ABB RobotStudio station: comportamiento1.rspag

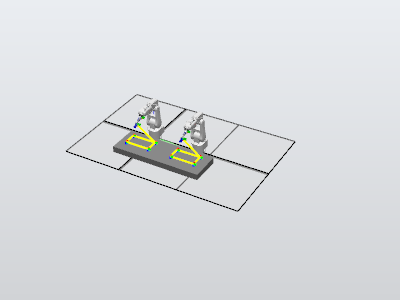
--- station ---
Station comportamiento1 (saved by RobotStudio 25.1.11133.0)
Controller IRB120_3_58_1, task T_ROB1: task frame (RAPID world) sits at (0, 800, 0) mm in the station
Controller IRB120_3_58
  mechanical unit ROB_1: IRB120_3_58__01, 6 joints, base frame (0, 0, 0) mm
Controller IRB120_3_58_1
  mechanical unit ROB_1: IRB120_3_58__02, 6 joints, base frame (0, 0, 0) mm
Layout (positions relative to the parent item):
  - IRB120_3_58__01 [mechanism, from %ABB.RobotStudio.Models.IRB120%\IRB120_3_58_G_01.rslib] at (0, 0, 0) mm; joint values [0, 0, 0, 0, 0.5236, 0] (rad or m)
  - IRB120_3_58__02 [mechanism, from %ABB.RobotStudio.Models.IRB120%\IRB120_3_58_G_01.rslib] at (0, 800, 0) mm; joint values [0, 0, 0, 0, 0.5236, 0] (rad or m)
  - SC_VentosaD50__1 [smart component, from Components\SC_VentosaD50.rslib] at (364.35, 0, 594) mm, rotated rx 180 ry 60 rz 180 deg
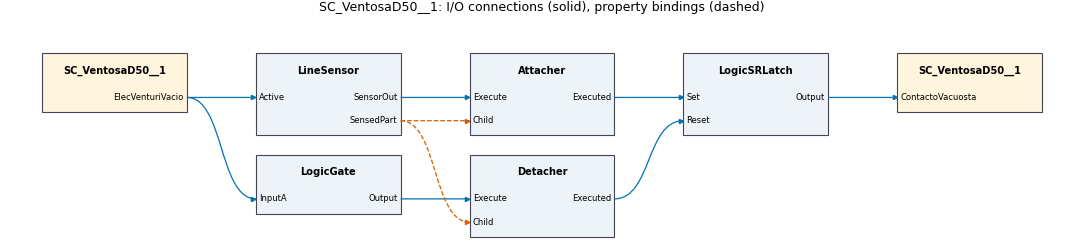
      connections:
        SC_VentosaD50__1.ElecVenturiVacio -> LineSensor.Active
        LineSensor.SensorOut -> Attacher.Execute
        Attacher.Executed -> LogicSRLatch.Set
        LogicSRLatch.Output -> SC_VentosaD50__1.ContactoVacuostato
        SC_VentosaD50__1.ElecVenturiVacio -> LogicGate.InputA
        LogicGate.Output -> Detacher.Execute
        Detacher.Executed -> LogicSRLatch.Reset
        LineSensor.SensedPart => Attacher.Child
        LineSensor.SensedPart => Detacher.Child
    - ToolVentosaD50 [mechanism, from Components\SC_VentosaD50.rslib] at (0, 0, 0) mm
    - Attacher [smart component, from Components\Attacher.rslib]
        properties: Parent=ToolVentosaD50; Flange=0; Child=(none); Mount=false; Offset=[0 0 0]; Orientation=[0 0 0]
    - Detacher [smart component, from Components\Detacher.rslib]
        properties: Child=(none); KeepPosition=true
    - LineSensor [smart component, from Components\LineSensor.rslib] at (0, 0, 126) mm
        properties: Start=[0 0 0]; End=[0 0 0.015]; Radius=0.001; SensedPart=(none); SensedPoint=[0 0 0]; Length=0.015; Tag=(none); SenseMultiple=false
      - _sensorPart_ [part], size 2 x 2 x 15 mm
    - LogicGate [smart component, from Components\LogicGate.rslib]
        properties: Operator=NOT; Delay=0
    - LogicSRLatch [smart component, from Components\LogicSRLatch.rslib]
  - SC_VentosaD50__2 [smart component, from Components\SC_VentosaD50.rslib] at (364.35, 800, 594) mm, rotated rx 180 ry 60 rz 180 deg
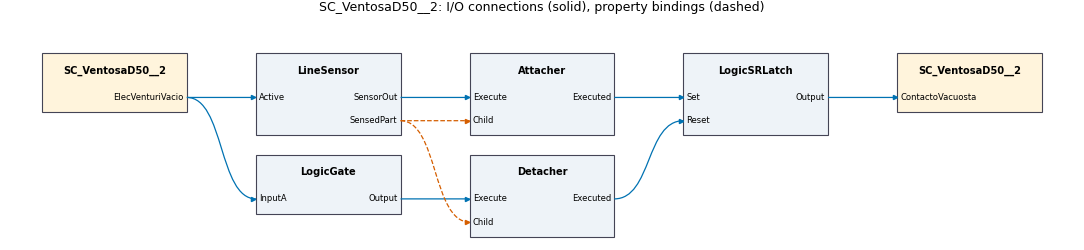
      connections:
        SC_VentosaD50__2.ElecVenturiVacio -> LineSensor.Active
        LineSensor.SensorOut -> Attacher.Execute
        Attacher.Executed -> LogicSRLatch.Set
        LogicSRLatch.Output -> SC_VentosaD50__2.ContactoVacuostato
        SC_VentosaD50__2.ElecVenturiVacio -> LogicGate.InputA
        LogicGate.Output -> Detacher.Execute
        Detacher.Executed -> LogicSRLatch.Reset
        LineSensor.SensedPart => Attacher.Child
        LineSensor.SensedPart => Detacher.Child
    - ToolVentosaD50 [mechanism, from Components\SC_VentosaD50.rslib] at (0, 0, 0) mm
    - Attacher [smart component, from Components\Attacher.rslib]
        properties: Parent=ToolVentosaD50; Flange=0; Child=(none); Mount=false; Offset=[0 0 0]; Orientation=[0 0 0]
    - Detacher [smart component, from Components\Detacher.rslib]
        properties: Child=(none); KeepPosition=true
    - LineSensor [smart component, from Components\LineSensor.rslib] at (0, 0, 126) mm
        properties: Start=[0 0 0]; End=[0 0 0.015]; Radius=0.001; SensedPart=(none); SensedPoint=[0 0 0]; Length=0.015; Tag=(none); SenseMultiple=false
      - _sensorPart_ [part], size 2 x 2 x 15 mm
    - LogicGate [smart component, from Components\LogicGate.rslib]
        properties: Operator=NOT; Delay=0
    - LogicSRLatch [smart component, from Components\LogicSRLatch.rslib]
  - Mesa de Trabajo [part], size 500 x 1500 x 100 mm
Attachment: SC_VentosaD50__1 is attached to IRB120_3_58__01 / Link6
Attachment: SC_VentosaD50__2 is attached to IRB120_3_58__02 / Link6

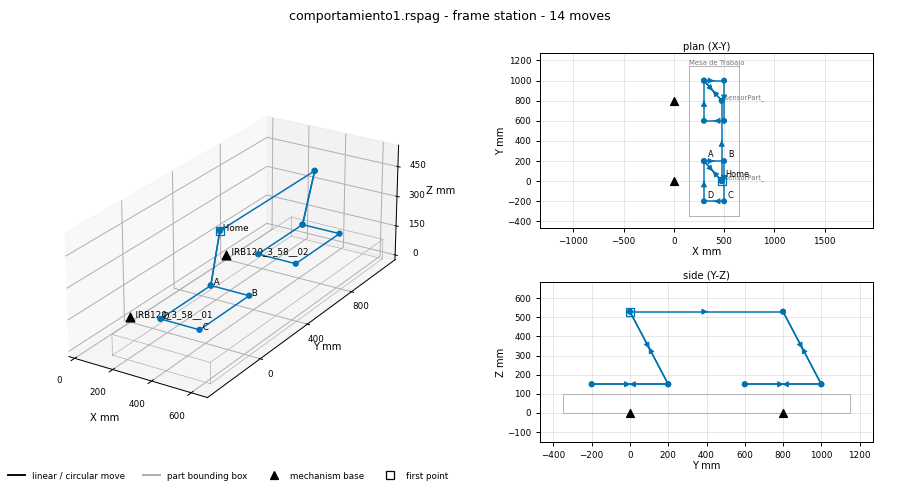
[picture p0: tool path of comportamiento1.rspag in frame station, 14 of 14 moves have a stored position in this frame; points joined in program order, loops and branches not executed]
--- Controller Data/IRB120_3_58/RAPID/TASK1/PROGMOD/CalibData.mod ---
MODULE CalibData
    PERS tooldata TCP_ToolVentosaD50:=[TRUE,[[0,0,129.5],[1,0,0,0]],[1,[0,0,1],[1,0,0,0],0,0,0]];
ENDMODULE

--- Controller Data/IRB120_3_58/RAPID/TASK1/PROGMOD/Module1.mod ---
MODULE Module1
    CONST robtarget Home:=[[476.504118863,0,529.25],[0.5,0,0.866025404,0],[0,0,0,0],[9E+09,9E+09,9E+09,9E+09,9E+09,9E+09]];
    CONST robtarget A:=[[300,200,150],[0,0,1,0],[0,0,0,0],[9E+09,9E+09,9E+09,9E+09,9E+09,9E+09]];
    CONST robtarget B:=[[500,200,150],[0,0,1,0],[0,0,0,0],[9E+09,9E+09,9E+09,9E+09,9E+09,9E+09]];
    CONST robtarget C:=[[500,-200,150],[0,0,1,0],[0,0,0,0],[9E+09,9E+09,9E+09,9E+09,9E+09,9E+09]];
    CONST robtarget D:=[[300,-200,150],[0,0,1,0],[0,0,0,0],[9E+09,9E+09,9E+09,9E+09,9E+09,9E+09]];
!***********************************************************
    !
    ! M?dulo:  Module1
    !
    ! Descripción:
    !   <Introduzca la descripción aquí>
    !
    ! Autor: Miguel
    !
    ! Versión: 1.0
    !
    !***********************************************************


    !***********************************************************
    !
    ! Procedimiento Main
    !
    !   Este es el punto de entrada de su programa
    !
    !***********************************************************
    PROC main()
        Path;
    ENDPROC
    PROC Path()
        MoveL Home,v500,fine,TCP_ToolVentosaD50\WObj:=wobj0;
        MoveL A,v500,fine,TCP_ToolVentosaD50\WObj:=wobj0;
        MoveL B,v500,fine,TCP_ToolVentosaD50\WObj:=wobj0;
        MoveL C,v500,fine,TCP_ToolVentosaD50\WObj:=wobj0;
        MoveL D,v500,fine,TCP_ToolVentosaD50\WObj:=wobj0;
        MoveL A,v500,fine,TCP_ToolVentosaD50\WObj:=wobj0;
        MoveL Home,v500,fine,TCP_ToolVentosaD50\WObj:=wobj0;
    ENDPROC
ENDMODULE

--- Controller Data/IRB120_3_58_1/RAPID/TASK1/PROGMOD/Module1.mod ---
MODULE Module1
    CONST robtarget Home:=[[476.504118863,0,529.25],[0.5,0,0.866025404,0],[0,0,0,0],[9E+09,9E+09,9E+09,9E+09,9E+09,9E+09]];
    CONST robtarget A:=[[300,200,150],[0,0,1,0],[0,0,0,0],[9E+09,9E+09,9E+09,9E+09,9E+09,9E+09]];
    CONST robtarget C:=[[500,-200,150],[0,0,1,0],[0,0,0,0],[9E+09,9E+09,9E+09,9E+09,9E+09,9E+09]];
    CONST robtarget D:=[[300,-200,150],[0,0,1,0],[0,0,0,0],[9E+09,9E+09,9E+09,9E+09,9E+09,9E+09]];
    CONST robtarget B:=[[500,200,150],[0,0,1,0],[0,0,0,0],[9E+09,9E+09,9E+09,9E+09,9E+09,9E+09]];
!***********************************************************
    !
    ! M?dulo:  Module1
    !
    ! Descripción:
    !   <Introduzca la descripción aquí>
    !
    ! Autor: Miguel Ferrer
    !
    ! Versión: 1.0
    !
    !***********************************************************


    !***********************************************************
    !
    ! Procedimiento Main
    !
    !   Este es el punto de entrada de su programa
    !
    !***********************************************************
    PROC main()
        Path;
    ENDPROC
    PROC Path()
        MoveL Home,v500,fine,TCP_ToolVentosaD50\WObj:=wobj0;
        MoveL A,v500,fine,TCP_ToolVentosaD50\WObj:=wobj0;
        MoveL B,v500,fine,TCP_ToolVentosaD50\WObj:=wobj0;
        MoveL C,v500,fine,TCP_ToolVentosaD50\WObj:=wobj0;
        MoveL D,v500,fine,TCP_ToolVentosaD50\WObj:=wobj0;
        MoveL A,v500,fine,TCP_ToolVentosaD50\WObj:=wobj0;
        MoveL Home,v500,fine,TCP_ToolVentosaD50\WObj:=wobj0;
    ENDPROC
ENDMODULE
